// TIA Portal project "cash register" (V16)

(* hardware
DEVICE "S7-1200 station_1"  S7-1200 Station
   slot 0: "Rack_0"  S7-1200 Rack  Rack  V1.0
   slot 1: "PLC_1"  CPU 1214C DC/DC/DC  6ES7 214-1AE30-0XB0  V2.2
   slot 3: "AQ 1x12BIT_1"  AQ1 signal board  6ES7 232-4HA30-0XB0  V1.0
*)

// ===== PLC "PLC_1"  CPU 1214C DC/DC/DC =====

VAR_GLOBAL   // PLC tag table "Default tag table"
   "dog" AT %M0.0 : Bool;
   "on" AT %M0.1 : Bool;
   "hotdog" AT %M0.2 : Bool;
   "drink" AT %M0.3 : Bool;
   "chicken nuggets" AT %M0.4 : Bool;
   "burger" AT %M0.5 : Bool;
   "new_hotdog" AT %MD2 : DInt;
   "Cancel_Last" AT %M6.0 : Bool;
   "total_hotdog" AT %M122.0 : LReal;
   "new_order" AT %M12.0 : Bool;
   "hotdog_sub" AT %MD14 : DInt;
   "hotdog_last" AT %M18.0 : Bool;
   "drink_sub" AT %MD20 : DInt;
   "new_drink" AT %MD24 : DInt;
   "total_drink" AT %M114.0 : LReal;
   "drink_last" AT %M32.0 : Bool;
   "chick_sub" AT %MD34 : DInt;
   "new_chick" AT %MD38 : DInt;
   "total_chick" AT %M106.0 : LReal;
   "chick_last" AT %M46.0 : Bool;
   "burger_sub" AT %MD48 : DInt;
   "new_burger" AT %MD52 : DInt;
   "total_burger" AT %M98.0 : LReal;
   "burger_last" AT %M60.0 : Bool;
   "fries" AT %M60.1 : Bool;
   "fries_sub" AT %MD62 : DInt;
   "new_fry" AT %MD66 : DInt;
   "total_fries" AT %M90.0 : LReal;
   "fries_last" AT %M74.0 : Bool;
   "Total" AT %M74.1 : Bool;
   "total_price" AT %M82.0 : LReal;
   "Tax" AT %M80.0 : Bool;
   "new_order_button" AT %M0.6 : Bool;
   "Cancel_button" AT %M0.7 : Bool;
END_VAR

// folder: System blocks/Program resources

DATA_BLOCK "hotdog_counter"   // DB1
{ S7_Optimized_Access := 'TRUE' }
AUTHOR : Simatic
FAMILY : IEC
NAME : CNTR
VERSION : 1.0
// stored: InstanceOfName IEC_COUNTER
"IEC_COUNTER"
BEGIN
END_DATA_BLOCK

DATA_BLOCK "drink_counter"   // DB2
{ S7_Optimized_Access := 'TRUE' }
AUTHOR : Simatic
FAMILY : IEC
NAME : CNTR
VERSION : 1.0
// stored: InstanceOfName IEC_COUNTER
"IEC_COUNTER"
BEGIN
END_DATA_BLOCK

DATA_BLOCK "hotdog_down"   // DB3
{ S7_Optimized_Access := 'TRUE' }
AUTHOR : Simatic
FAMILY : IEC
NAME : CNTR
VERSION : 1.0
// stored: InstanceOfName IEC_COUNTER
"IEC_COUNTER"
BEGIN
END_DATA_BLOCK

DATA_BLOCK "drink_down"   // DB4
{ S7_Optimized_Access := 'TRUE' }
AUTHOR : Simatic
FAMILY : IEC
NAME : CNTR
VERSION : 1.0
// stored: InstanceOfName IEC_COUNTER
"IEC_COUNTER"
BEGIN
END_DATA_BLOCK

DATA_BLOCK "chick_counter"   // DB5
{ S7_Optimized_Access := 'TRUE' }
AUTHOR : Simatic
FAMILY : IEC
NAME : CNTR
VERSION : 1.0
// stored: InstanceOfName IEC_COUNTER
"IEC_COUNTER"
BEGIN
END_DATA_BLOCK

DATA_BLOCK "chick_down"   // DB6
{ S7_Optimized_Access := 'TRUE' }
AUTHOR : Simatic
FAMILY : IEC
NAME : CNTR
VERSION : 1.0
// stored: InstanceOfName IEC_COUNTER
"IEC_COUNTER"
BEGIN
END_DATA_BLOCK

DATA_BLOCK "burger_counter"   // DB7
{ S7_Optimized_Access := 'TRUE' }
AUTHOR : Simatic
FAMILY : IEC
NAME : CNTR
VERSION : 1.0
// stored: InstanceOfName IEC_COUNTER
"IEC_COUNTER"
BEGIN
END_DATA_BLOCK

DATA_BLOCK "burger_down"   // DB8
{ S7_Optimized_Access := 'TRUE' }
AUTHOR : Simatic
FAMILY : IEC
NAME : CNTR
VERSION : 1.0
// stored: InstanceOfName IEC_COUNTER
"IEC_COUNTER"
BEGIN
END_DATA_BLOCK

DATA_BLOCK "fry_counter"   // DB9
{ S7_Optimized_Access := 'TRUE' }
AUTHOR : Simatic
FAMILY : IEC
NAME : CNTR
VERSION : 1.0
// stored: InstanceOfName IEC_COUNTER
"IEC_COUNTER"
BEGIN
END_DATA_BLOCK

DATA_BLOCK "fries_down"   // DB10
{ S7_Optimized_Access := 'TRUE' }
AUTHOR : Simatic
FAMILY : IEC
NAME : CNTR
VERSION : 1.0
// stored: InstanceOfName IEC_COUNTER
"IEC_COUNTER"
BEGIN
END_DATA_BLOCK

// folder: (top level)

ORGANIZATION_BLOCK "Main"   // OB1, LAD, ProgramCycle
TITLE = "Main Program Sweep (Cycle)"
{ S7_Optimized_Access := 'TRUE' }
VERSION : 0.1
BEGIN

REGION Network 1
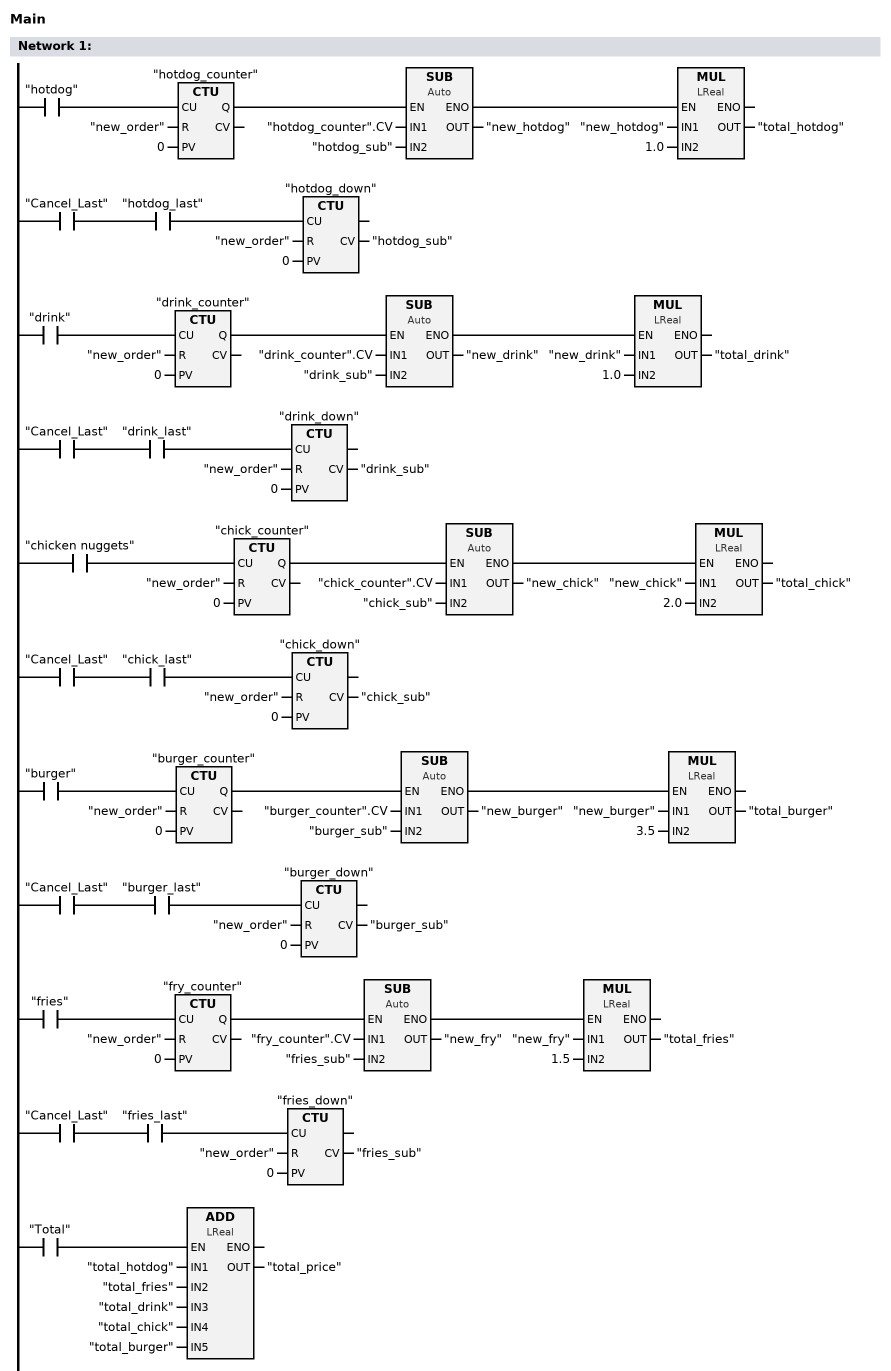
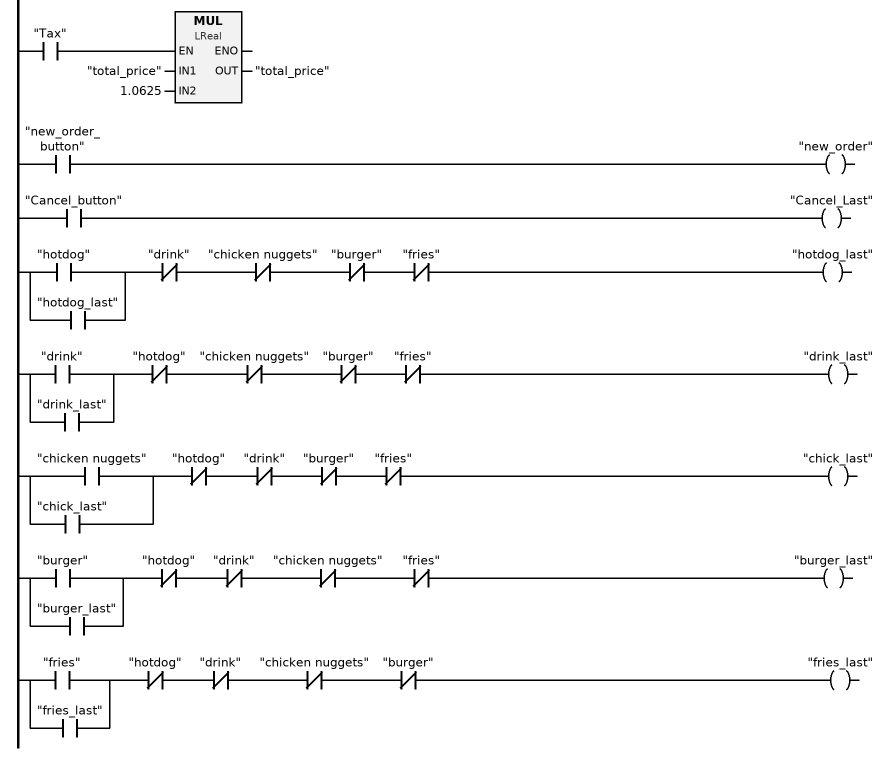
   // ENO of a box is taken as its EN; it also drops when the box reports an error
   "hotdog_counter".CTU(CU := "hotdog", R := "new_order", PV := 0);
   IF "hotdog_counter".Q THEN
       "new_hotdog" := "hotdog_counter".CV - "hotdog_sub";
       "total_hotdog" := "new_hotdog" * 1.0;
   END_IF;
   "hotdog_down".CTU(CU := "Cancel_Last" AND "hotdog_last", R := "new_order", PV := 0, CV => "hotdog_sub");
   "drink_counter".CTU(CU := "drink", R := "new_order", PV := 0);
   IF "drink_counter".Q THEN
       "new_drink" := "drink_counter".CV - "drink_sub";
       "total_drink" := "new_drink" * 1.0;
   END_IF;
   "drink_down".CTU(CU := "Cancel_Last" AND "drink_last", R := "new_order", PV := 0, CV => "drink_sub");
   "chick_counter".CTU(CU := "chicken nuggets", R := "new_order", PV := 0);
   IF "chick_counter".Q THEN
       "new_chick" := "chick_counter".CV - "chick_sub";
       "total_chick" := "new_chick" * 2.0;
   END_IF;
   "chick_down".CTU(CU := "Cancel_Last" AND "chick_last", R := "new_order", PV := 0, CV => "chick_sub");
   "burger_counter".CTU(CU := "burger", R := "new_order", PV := 0);
   IF "burger_counter".Q THEN
       "new_burger" := "burger_counter".CV - "burger_sub";
       "total_burger" := "new_burger" * 3.5;
   END_IF;
   "burger_down".CTU(CU := "Cancel_Last" AND "burger_last", R := "new_order", PV := 0, CV => "burger_sub");
   "fry_counter".CTU(CU := "fries", R := "new_order", PV := 0);
   IF "fry_counter".Q THEN
       "new_fry" := "fry_counter".CV - "fries_sub";
       "total_fries" := "new_fry" * 1.5;
   END_IF;
   "fries_down".CTU(CU := "Cancel_Last" AND "fries_last", R := "new_order", PV := 0, CV => "fries_sub");
   IF "Total" THEN
       "total_price" := "total_hotdog" + "total_fries" + "total_drink" + "total_chick" + "total_burger";
   END_IF;
   IF "Tax" THEN "total_price" := "total_price" * 1.0625; END_IF;
   "new_order" := "new_order_button";
   "Cancel_Last" := "Cancel_button";
   "hotdog_last" := ("hotdog" OR "hotdog_last") AND NOT "drink" AND NOT "chicken nuggets" AND NOT "burger" AND NOT "fries";
   "drink_last" := ("drink" OR "drink_last") AND NOT "hotdog" AND NOT "chicken nuggets" AND NOT "burger" AND NOT "fries";
   "chick_last" := ("chicken nuggets" OR "chick_last") AND NOT "hotdog" AND NOT "drink" AND NOT "burger" AND NOT "fries";
   "burger_last" := ("burger" OR "burger_last") AND NOT "hotdog" AND NOT "drink" AND NOT "chicken nuggets" AND NOT "fries";
   "fries_last" := ("fries" OR "fries_last") AND NOT "hotdog" AND NOT "drink" AND NOT "chicken nuggets" AND NOT "burger";
END_REGION
END_ORGANIZATION_BLOCK